(* CoDeSys 2.3.9.37 project: Cap3_2.pro *)
(* Libraries: Standard.lib 4.10.05 12:14:46 *)

(* POU PLC_PRG, LD *)
PROGRAM PLC_PRG
VAR
	P: BOOL;
	M: BOOL;
	Motor: BOOL;
END_VAR
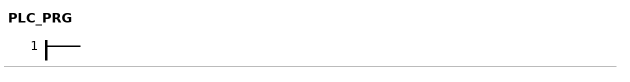
_LD_ (* Ladder Diagram *)
NETWORK 1
	*
_END_LD_
(* the same logic as Structured Text *)
(* Network 1 *)
END_PROGRAM

(* Visualisation Botonera
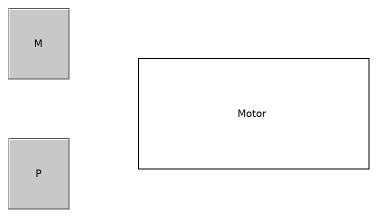
rounded rectangle at (200,80)-(431,191): text "Motor"; alarm colour if PLC_PRG.Motor
button at (70,30)-(131,101): text "M"; taps PLC_PRG.M
button at (70,160)-(131,231): text "P"; taps PLC_PRG.P
*)
